// TIA Portal V20 export
FUNCTION_BLOCK "FB_MiscPLC_IHM_ISO"   // FB50, SCL
{ S7_Optimized_Access := 'TRUE' }
// stored: MemoryReserve 100, SetENOAutomatically false
   VAR
      sTransferSelData { S7_SetPoint := 'True'} : Array[0..11] of Byte;
      sTransferActData : Array[0..11] of Byte;
      sUpdate_PLC_ISO_Values : Bool;
      sRT_bStopAfterEmptying : R_TRIG;
      sRT_CNCModeReq { S7_SetPoint := 'True'} : R_TRIG;
   END_VAR
   VAR_TEMP
      tLoop : Int;
      tTransferSelDataError : Int;
      tTransferSelDataErrCode : Array[0..11] of Int;
   END_VAR
BEGIN
   REGION Description header 
       //==================================================================================
       // POSALUX Swiss SA / (C) Copyright 2025
       //----------------------------------------------------------------------------------
       // Title: 
       // Comment/Function: 
       // Author: Fabien WALDT
       // Engineering: TIA Portal v17
       //----------------------------------------------------------------------------------
       // Change log table:
       // Version  | Date     | Expert in charge | Changes applied
       // ---------|----------|------------------|-----------------------------------------
       // 00.00.01 | 20250423 | WFA              | First released version
       // =================================================================================
   END_REGION

   REGION Byte 960
       // Bit 0
       "DB_PLC_ISO_IHM".WarmUpOn := "LBP_AlarmMsgs".UserA[0].A70UUxx[35];

       // Bit 1
       "DB_PLC_ISO_IHM".KeyLaserOn := "DB_DataFromSafety".iKeyLaserOn;

       // Bit 2
       "DB_PLC_ISO_IHM".KeySaveParameters := "DB_McpKeyboardSignals".sK3_KeySaveParam.sKeySWToggleStatus;
       "DB_McpKeyboardSignals".sK3_KeySaveParam.sLedSWStatus := "DB_McpKeyboardSignals".sK3_KeySaveParam.sKeySWToggleStatus;

       // Bit 3
       // STOP_PROG_RUN est nommé bStopAfterEmptying dans PLC
       #sRT_bStopAfterEmptying(CLK := "DB_WorkingModes".sEmptying AND "DB_PartManagement".sPosition.sMachineEmpty);
       IF #sRT_bStopAfterEmptying.Q THEN
           "DB_PLC_ISO_IHM".bStopAfterEmptying := TRUE;
           "LBP_AlarmMsgs".UserA[0].A70UUxx[59] := TRUE;
           "DB_WorkingModes".sEmptying := FALSE;
           "DB_LoaderShuttle1".sMain.iJobReq := FALSE;
           "DB_LoaderShuttle2".sMain.iJobReq := FALSE;
       ELSIF "LBP_Chan1".E_ChanReset THEN
           "DB_PLC_ISO_IHM".bStopAfterEmptying := FALSE;
       END_IF;

       // Bit 4
       "DB_PLC_ISO_IHM".Chan1_running := "DB_CycleStartStop".sChan1Start;

       // Bit 5
       "DB_PLC_ISO_IHM".Chan2_running := FALSE;

       // Bit 6
       "DB_PLC_ISO_IHM".Chan3_running := FALSE;

       // Bit 7
       "DB_PLC_ISO_IHM".Chan4_running := FALSE;
   END_REGION

   REGION Byte 961
       // Bit 0
       "DB_PLC_ISO_IHM".StopAtNextReq := "DB_CycleStartStop".sResquestStopNextCycle;

       // Bit 1
       "DB_PLC_ISO_IHM".AllChanStop := NOT "DB_CycleStartStop".sChan1Start;

       // Bit 2
       "DB_PLC_ISO_IHM".LoaderAutomaticMode := "DB_WorkingModes".sAuto;

       // Bit 3
       "DB_PLC_ISO_IHM".LoaderManualMode := "DB_WorkingModes".sSemiAuto;

       // Bit 4 (NOT USED ON FL0125)
       "DB_PLC_ISO_IHM".NoCameraPresent := "DB_PLC_ISO_IHM".NoCameraPresent;

       // Bit 5 (NOT USED ON FL0125)
       "DB_PLC_ISO_IHM".PremeasureZexists := "DB_PLC_ISO_IHM".PremeasureZexists;

       // Bit 6 (NOT USED ON FL0125)
       "DB_PLC_ISO_IHM".PremeasureCexists := "DB_PLC_ISO_IHM".PremeasureCexists;

       // Bit 7
       "DB_PLC_ISO_IHM".PLCFunctNotFinished :=
       "DB_LoaderFixtureMain".sBlowingNotFinished
       OR "DB_LoaderFixtureMain".sLoadingNotFinished
       OR "DB_LoaderFixtureMain".sUnloadingNotFinished
       OR "DB_LoaderFixtureMain".sReleaseNotFinished
       OR "DB_LoaderFixtureMain".sV_InitNotFinished
       OR "DB_LoaderFixtureMain".sW_InitNotFinished;
   END_REGION

   REGION Byte 962
       // Bit 0
       // CAN_CHANGE_PART_LOADER_1 est nommé StartChangePart_station1 dans PLC
       #sRT_CNCModeReq(CLK := "DB_LoaderAxis".iCNCModeReq);

       IF #sRT_CNCModeReq.Q AND NOT "DB_PartManagement".sPosition.sMachineEmpty THEN
           "DB_PLC_ISO_IHM".StartChangePart_station1 := TRUE;
       ELSIF "LBP_Chan1".MDyn[76] THEN
           "DB_PLC_ISO_IHM".StartChangePart_station1 := FALSE;
       END_IF;

       // Bit 1
       "DB_PLC_ISO_IHM".StartCheckPart_fixture1 := "DB_PLC_ISO_IHM".StartCheckPart_fixture1;

       // Bit 2
       "DB_PLC_ISO_IHM".Loader1PartLoad := "DB_PartManagement".sPosition.sGripper.Undrilled.Presence.Part AND "DB_PartManagement".sPosition.sGripper.Undrilled.Presence.BW;

       // Bit 3
       "DB_PLC_ISO_IHM".Loader1PartUnload := "DB_PartManagement".sPosition.sGripper.Drilled.Presence.Part;

       // Bit 4
       "DB_PLC_ISO_IHM".Loader1ShiftLoad := "DB_PLC_ISO_IHM".Loader1ShiftLoad;

       // Bit 5
       "DB_PLC_ISO_IHM".Loader1ShiftUnload := "DB_PLC_ISO_IHM".Loader1ShiftUnload;

       // Bit 6
       "DB_PLC_ISO_IHM".Loader1LoadOpened := "DB_PLC_ISO_IHM".Loader1LoadOpened;

       // Bit 7
       "DB_PLC_ISO_IHM".Loader1UnloadOpened := "DB_PLC_ISO_IHM".Loader1UnloadOpened;
   END_REGION

   REGION Byte 963
       // Bit 0
       "DB_PLC_ISO_IHM".PartOnFixture1 := "DB_GestionFixture".sFixturePartControl.oGoodPart
               OR "DB_PartManagement".sPosition.sFixture.Undrilled.Presence.Part
               OR "DB_PartManagement".sPosition.sFixture.Drilled.Presence.Part;

       // Bit 1
       "DB_PLC_ISO_IHM".MasterOnFixture1 := "DB_PLC_ISO_IHM".MasterOnFixture1;

       // Bit 2
       "DB_PLC_ISO_IHM".StartChangePart_station2 := "DB_PLC_ISO_IHM".StartChangePart_station2;

       // Bit 3
       "DB_PLC_ISO_IHM".StartCheckPart_fixture2 := "DB_PLC_ISO_IHM".StartCheckPart_fixture2;

       // Bit 4
       "DB_PLC_ISO_IHM".Loader2PartLoad := "DB_PLC_ISO_IHM".Loader2PartLoad;

       // Bit 5
       "DB_PLC_ISO_IHM".Loader2PartUnload := "DB_PLC_ISO_IHM".Loader2PartUnload;

       // Bit 6
       "DB_PLC_ISO_IHM".Loader2ShiftLoad := "DB_PLC_ISO_IHM".Loader2ShiftLoad;

       // Bit 7
       "DB_PLC_ISO_IHM".Loader2ShiftUnload := "DB_PLC_ISO_IHM".Loader2ShiftUnload;
   END_REGION

   REGION Byte 964
       // Bit 0
       "DB_PLC_ISO_IHM".Loader2LoadOpened := "DB_PLC_ISO_IHM".Loader2LoadOpened;

       // Bit 1
       "DB_PLC_ISO_IHM".Loader2UnloadOpened := "DB_PLC_ISO_IHM".Loader2UnloadOpened;

       // Bit 2 
       "DB_PLC_ISO_IHM".PartOnFixture2 := "DB_PLC_ISO_IHM".PartOnFixture2;

       // Bit 3 (NOT USED ON FL0125)
       "DB_PLC_ISO_IHM".MasterOnFixture2 := "DB_PLC_ISO_IHM".MasterOnFixture2;

       // Bit 4 (NOT USED ON FL0125)
       "DB_PLC_ISO_IHM".StartChangePart_station3 := "DB_PLC_ISO_IHM".StartChangePart_station3;

       // Bit 5 (NOT USED ON FL0125)
       "DB_PLC_ISO_IHM".StartCheckPart_fixture3 := "DB_PLC_ISO_IHM".StartCheckPart_fixture3;

       // Bit 6 (NOT USED ON FL0125)
       "DB_PLC_ISO_IHM".Loader3PartLoad := "DB_PLC_ISO_IHM".Loader3PartLoad;

       // Bit 7 (NOT USED ON FL0125)
       "DB_PLC_ISO_IHM".Loader3PartUnload := "DB_PLC_ISO_IHM".Loader3PartUnload;
   END_REGION

   REGION Byte 965
       // Bit 0 (NOT USED ON FL0125)
       "DB_PLC_ISO_IHM".Loader3ShiftLoad := "DB_PLC_ISO_IHM".Loader3ShiftLoad;

       // Bit 1 (NOT USED ON FL0125)
       "DB_PLC_ISO_IHM".Loader3ShiftUnload := "DB_PLC_ISO_IHM".Loader3ShiftUnload;

       // Bit 2 (NOT USED ON FL0125)
       "DB_PLC_ISO_IHM".Loader3LoadOpened := "DB_PLC_ISO_IHM".Loader3LoadOpened;

       // Bit 3
       "DB_PLC_ISO_IHM".Loader3UnloadOpened := "DB_PLC_ISO_IHM".Loader3UnloadOpened;

       // Bit 4
       "DB_PLC_ISO_IHM".PartOnFixture3 := "DB_PLC_ISO_IHM".PartOnFixture3;

       // Bit 5 (NOT USED ON FL0125)
       "DB_PLC_ISO_IHM".MasterOnFixture3 := "DB_PLC_ISO_IHM".MasterOnFixture3;

       // Bit 6 (NOT USED ON FL0125)
       "DB_PLC_ISO_IHM".Part_KO_go_outside_mach := "DB_PLC_ISO_IHM".Part_KO_go_outside_mach;

       // Bit 7 (NOT USED ON FL0125)
       "DB_PLC_ISO_IHM".MasterOnMachine := "DB_PLC_ISO_IHM".MasterOnMachine;
   END_REGION

   REGION Word 968
       "DB_PLC_ISO_IHM".WarmUpTime := "DB_PLC_ISO_IHM".WarmUpTime;
   END_REGION

   REGION Byte 970
       // Bit 0
       "DB_PLC_ISO_IHM".Stop_For_BackWall_Wear_1 := "DB_PLC_ISO_IHM".Stop_For_BackWall_Wear_1;

       // Bit 1
       "DB_PLC_ISO_IHM".Stop_For_BackWall_Wear_2 := "DB_PLC_ISO_IHM".Stop_For_BackWall_Wear_2;

       // Bit 2
       "DB_PLC_ISO_IHM".Cleaning_Station_1 := "DB_PLC_ISO_IHM".Cleaning_Station_1;

       // Bit 3
       "DB_PLC_ISO_IHM".Cleaning_Station_2 := "DB_PLC_ISO_IHM".Cleaning_Station_2;

       // Bit 4
       "DB_PLC_ISO_IHM".Cleaning_Backwall_1 := "DB_PLC_ISO_IHM".Cleaning_Backwall_1;

       // Bit 5
       "DB_PLC_ISO_IHM".Cleaning_Backwall_2 := "DB_PLC_ISO_IHM".Cleaning_Backwall_2;

       // Bit 6
       "DB_PLC_ISO_IHM".Shutter_laser_closed := "DB_DigitalInputs".sShutterClosed.sSWStatus OR
            NOT "DB_DataFromSafety".iKeyLaserOn;

       // Bit 7
       "DB_PLC_ISO_IHM".Pressure_Stop_Machine := "DB_PLC_ISO_IHM".Pressure_Stop_Machine;
   END_REGION

   REGION Byte 971  
       // Bit 0
       IF "LBP_Chan1".MDyn[68] OR "DB_Scanner".sScannerComm.oGoodPart THEN
           "DB_PLC_ISO_IHM".BadPartOnFixture := FALSE;
       ELSIF "DB_BadPartOnFixture".BadPartOnFixture
           OR "DB_GestionFixture".sFixturePartControl.oBadpart
           OR "DB_Scanner".sScannerComm.oBadPart THEN
               "DB_PLC_ISO_IHM".BadPartOnFixture := TRUE;
       END_IF;

       // Bit 1 (NOT USED ON FL0125)
       "DB_PLC_ISO_IHM".Reserve12 := "DB_PLC_ISO_IHM".Reserve12;

       // Bit 2 (NOT USED ON FL0125)
       "DB_PLC_ISO_IHM".Reserve13 := "DB_PLC_ISO_IHM".Reserve13;

       // Bit 3 (NOT USED ON FL0125)
       "DB_PLC_ISO_IHM".Reserve14 := "DB_PLC_ISO_IHM".Reserve14;

       // Bit 4 (NOT USED ON FL0125)
       "DB_PLC_ISO_IHM".Reserve15 := "DB_PLC_ISO_IHM".Reserve15;

       // Bit 5
       "DB_PLC_ISO_IHM".SemiAuto_RunEmpty := "DB_PLC_ISO_IHM".SemiAuto_RunEmpty;

       // Bit 6
       "DB_PLC_ISO_IHM"."SemiAuto_Unload_C-Fixture" := "DB_PLC_ISO_IHM"."SemiAuto_Unload_C-Fixture";

       // Bit 7 (NOT USED ON FL0125)
       "DB_PLC_ISO_IHM".Reserve18 := "DB_PLC_ISO_IHM".Reserve18;
   END_REGION

   REGION Transfert data PLC -> ISO

       FOR #tLoop := 0 TO 11 DO
           #sTransferActData[#tLoop] := PEEK(area := 16#84, dbNumber := 1302, byteOffset := #tLoop);
           IF #sTransferActData[#tLoop] <> #sTransferSelData[#tLoop] THEN
               #sUpdate_PLC_ISO_Values := TRUE;
               #sTransferSelData[#tLoop] := #sTransferActData[#tLoop];
           END_IF;
       END_FOR;

       // Transfert DB_PLC_ISO_IHM DWORD 0  

       // DEFINE PART_ON_FIXTURE_1         AS (($A_DBB[963] B_AND 1)==1)
       // DEFINE MASTER_ON_FIXTURE_1       AS (($A_DBB[963] B_AND 2)==2)
       // DEFINE CAN_CHANGE_PART_LOADER_2  AS (($A_DBB[963] B_AND 4)==4)
       // DEFINE CHECK_PART_FIXTURE_2      AS (($A_DBB[963] B_AND 8)==8)
       // DEFINE LOADER_2_PART_LOAD        AS (($A_DBB[963] B_AND 16)==16)
       // DEFINE LOADER_2_PART_UNLOAD      AS (($A_DBB[963] B_AND 32)==32)
       // DEFINE LOADER_2_SHIFT_LOAD       AS (($A_DBB[963] B_AND 64)==64)
       // DEFINE LOADER_2_SHIFT_UNLOAD     AS (($A_DBB[963] B_AND 128)==128)

       "LBP_TransferSelData"(Enable := #sUpdate_PLC_ISO_Values,
                             Funct := BYTE#16#04,
                             IVAR1 := 963,
                             IVAR2 := -1,
                             Error => #tTransferSelDataError.%X0,
                             ErrCode => #tTransferSelDataErrCode[0],
                             S7Var := #sTransferSelData[3]);

       // DEFINE CAN_CHANGE_PART_LOADER_1  AS (($A_DBB[962] B_AND 1)==1)
       // DEFINE CHECK_PART_FIXTURE_1      AS (($A_DBB[962] B_AND 2)==2)
       // DEFINE LOADER_1_PART_LOAD        AS (($A_DBB[962] B_AND 4)==4)
       // DEFINE LOADER_1_PART_UNLOAD      AS (($A_DBB[962] B_AND 8)==8)
       // DEFINE LOADER_1_SHIFT_LOAD       AS (($A_DBB[962] B_AND 16)==16)
       // DEFINE LOADER_1_SHIFT_UNLOAD     AS (($A_DBB[962] B_AND 32)==32)
       // DEFINE LOADER_1_LOAD_OPENED      AS (($A_DBB[962] B_AND 64)==64)
       // DEFINE LOADER_1_UNLOAD_OPENED    AS (($A_DBB[962] B_AND 128)==128)

       "LBP_TransferSelData"(Enable := #sUpdate_PLC_ISO_Values,
                             Funct := BYTE#16#04,
                             IVAR1 := 962,
                             IVAR2 := -1,
                             Error => #tTransferSelDataError.%X1,
                             ErrCode => #tTransferSelDataErrCode[1],
                             S7Var := #sTransferSelData[2]);

       // DEFINE STOP_AT_NEXT_REQ          AS (($A_DBB[961] B_AND 1)==1)
       // DEFINE ALL_CHAN_STOP             AS (($A_DBB[961] B_AND 2)==2)
       // DEFINE LOADER_MODE_AUTOMATIC     AS (($A_DBB[961] B_AND 4)==4)
       // DEFINE LOADER_MODE_MANUAL        AS (($A_DBB[961] B_AND 8)==8)
       // DEFINE MODE_WITH_LOADER          AS (($A_DBB[961] B_AND 12)>0)
       // DEFINE MODE_WITHOUT_LOADER       AS (($A_DBB[961] B_AND 12)==0)
       // DEFINE NO_CAMERA_PRESENT         AS (($A_DBB[961] B_AND 16)==16)
       // DEFINE PREMEASURE_Z_EXISTS       AS (($A_DBB[961] B_AND 32)==32)
       // DEFINE PREMEASURE_C_EXISTS       AS (($A_DBB[961] B_AND 64)==64)

       "LBP_TransferSelData"(Enable := #sUpdate_PLC_ISO_Values,
                             Funct := BYTE#16#04,
                             IVAR1 := 961,
                             IVAR2 := -1,
                             Error => #tTransferSelDataError.%X2,
                             ErrCode => #tTransferSelDataErrCode[2],
                             S7Var := #sTransferSelData[1]);

       // DEFINE WARM_UP_ON                AS (($A_DBB[960] B_AND 1)==1)
       // DEFINE KEY_LASER_ON              AS (($A_DBB[960] B_AND 2)==2)
       // DEFINE KEY_SAVE_PARAM            AS (($A_DBB[960] B_AND 4)==4)
       // DEFINE STOP_PROG_RUN             AS (($A_DBB[960] B_AND 8)==8)
       // DEFINE CHAN_1_RUNNING            AS (($A_DBB[960] B_AND 16)==16)
       // DEFINE CHAN_2_RUNNING            AS (($A_DBB[960] B_AND 32)==32)
       // DEFINE CHAN_3_RUNNING            AS (($A_DBB[960] B_AND 64)==64)
       // DEFINE CHAN_4_RUNNING            AS (($A_DBB[960] B_AND 128)==128)

       "LBP_TransferSelData"(Enable := #sUpdate_PLC_ISO_Values,
                             Funct := BYTE#16#04,
                             IVAR1 := 960,
                             IVAR2 := -1,
                             Error => #tTransferSelDataError.%X3,
                             ErrCode => #tTransferSelDataErrCode[3],
                             S7Var := #sTransferSelData[0]);

       // Transfert DB_PLC_ISO_IHM DWORD 4  


       "LBP_TransferSelData"(Enable := #sUpdate_PLC_ISO_Values,
                             Funct := BYTE#16#04,
                             IVAR1 := 967,
                             IVAR2 := -1,
                             Error => #tTransferSelDataError.%X4,
                             ErrCode => #tTransferSelDataErrCode[4],
                             S7Var := #sTransferSelData[7]);

       "LBP_TransferSelData"(Enable := #sUpdate_PLC_ISO_Values,
                             Funct := BYTE#16#04,
                             IVAR1 := 966,
                             IVAR2 := -1,
                             Error => #tTransferSelDataError.%X5,
                             ErrCode => #tTransferSelDataErrCode[5],
                             S7Var := #sTransferSelData[6]);

       // DEFINE LOADER_3_SHIFT_LOAD       AS (($A_DBB[965] B_AND 1)==1)
       // DEFINE LOADER_3_SHIFT_UNLOAD     AS (($A_DBB[965] B_AND 2)==2)
       // DEFINE LOADER_3_LOAD_OPENED      AS (($A_DBB[965] B_AND 4)==4)
       // DEFINE LOADER_3_UNLOAD_OPENED    AS (($A_DBB[965] B_AND 8)==8)
       // DEFINE PART_ON_FIXTURE_3         AS (($A_DBB[965] B_AND 16)==16)
       // DEFINE MASTER_ON_FIXTURE_3       AS (($A_DBB[965] B_AND 32)==32)
       // DEFINE PART_KO_GO_OUTSIDE        AS (($A_DBB[965] B_AND 64)==64)
       // DEFINE MASTER_ON_MACHINE         AS (($A_DBB[965] B_AND 128)==128)

       "LBP_TransferSelData"(Enable := #sUpdate_PLC_ISO_Values,
                             Funct := BYTE#16#04,
                             IVAR1 := 965,
                             IVAR2 := -1,
                             Error => #tTransferSelDataError.%X6,
                             ErrCode => #tTransferSelDataErrCode[6],
                             S7Var := #sTransferSelData[5]);

       // DEFINE LOADER_2_LOAD_OPENED      AS (($A_DBB[964] B_AND 1)==1)
       // DEFINE LOADER_2_UNLOAD_OPENED    AS (($A_DBB[964] B_AND 2)==2)
       // DEFINE PART_ON_FIXTURE_2         AS (($A_DBB[964] B_AND 4)==4)
       // DEFINE MASTER_ON_FIXTURE_2       AS (($A_DBB[964] B_AND 8)==8)
       // DEFINE CAN_CHANGE_PART_LOADER_3  AS (($A_DBB[964] B_AND 16)==16)
       // DEFINE CHECK_PART_FIXTURE_3      AS (($A_DBB[964] B_AND 32)==32)
       // DEFINE LOADER_3_PART_LOAD        AS (($A_DBB[964] B_AND 64)==64)
       // DEFINE LOADER_3_PART_UNLOAD      AS (($A_DBB[964] B_AND 128)==128)

       "LBP_TransferSelData"(Enable := #sUpdate_PLC_ISO_Values,
                             Funct := BYTE#16#04,
                             IVAR1 := 964,
                             IVAR2 := -1,
                             Error => #tTransferSelDataError.%X7,
                             ErrCode => #tTransferSelDataErrCode[7],
                             S7Var := #sTransferSelData[4]);

       // Transfert DB_PLC_ISO_IHM DWORD 8  

       // DEFINE SET_BAD_PART_ON_FIXTURE   AS (($A_DBB[971] B_AND 1)==1)
       // ;DEFINE     AS (($A_DBB[971] B_AND 2)==2)
       // ;DEFINE     AS (($A_DBB[971] B_AND 4)==4)
       // ;DEFINE     AS (($A_DBB[971] B_AND 8)==8)
       // ;DEFINE     AS (($A_DBB[971] B_AND 16)==16)
       // DEFINE SEMIAUTO_RUNEMPTY         AS (($A_DBB[971] B_AND 32)==32)
       // DEFINE SEMIAUTO_UNLOAD_C_FIXTURE AS (($A_DBB[971] B_AND 64)==64)
       // ;DEFINE     AS (($A_DBB[971] B_AND 128)==128

       "LBP_TransferSelData"(Enable := #sUpdate_PLC_ISO_Values,
                             Funct := BYTE#16#04,
                             IVAR1 := 971,
                             IVAR2 := -1,
                             Error => #tTransferSelDataError.%X8,
                             ErrCode => #tTransferSelDataErrCode[8],
                             S7Var := #sTransferSelData[11]);

       // DEFINE STOP_FOR_BACKWALL1_WEARED AS (($A_DBB[970] B_AND 1)==1)
       // DEFINE STOP_FOR_BACKWALL2_WEARED AS (($A_DBB[970] B_AND 2)==2)
       // DEFINE CLEANING_STATION1         AS (($A_DBB[970] B_AND 4)==4)
       // DEFINE CLEANING_STATION2         AS (($A_DBB[970] B_AND 8)==8)
       // DEFINE CLEANING_BACKWALL1        AS (($A_DBB[970] B_AND 16)==16)
       // DEFINE CLEANING_BACKWALL2        AS (($A_DBB[970] B_AND 32)==32)
       // DEFINE LASER_SHUTTER_CLOSED      AS (($A_DBB[970] B_AND 64)==64)
       // DEFINE NOT_COND_FOR_DRILL        AS (($A_DBB[970] B_AND 128)==128)

       "LBP_TransferSelData"(Enable := #sUpdate_PLC_ISO_Values,
                             Funct := BYTE#16#04,
                             IVAR1 := 970,
                             IVAR2 := -1,
                             Error => #tTransferSelDataError.%X9,
                             ErrCode => #tTransferSelDataErrCode[9],
                             S7Var := #sTransferSelData[10]);


       "LBP_TransferSelData"(Enable := #sUpdate_PLC_ISO_Values,
                             Funct := BYTE#16#04,
                             IVAR1 := 969,
                             IVAR2 := -1,
                             Error => #tTransferSelDataError.%X10,
                             ErrCode => #tTransferSelDataErrCode[10],
                             S7Var := #sTransferSelData[9]);

       // DEFINE WARM_UP_TIME              AS ($A_DBW[968])

       "LBP_TransferSelData"(Enable := #sUpdate_PLC_ISO_Values,
                             Funct := BYTE#16#04,
                             IVAR1 := 968,
                             IVAR2 := -1,
                             Error => #tTransferSelDataError.%X11,
                             ErrCode => #tTransferSelDataErrCode[11],
                             S7Var := #sTransferSelData[8]);

       IF #tTransferSelDataError = 0 THEN
           #sUpdate_PLC_ISO_Values := FALSE;
       END_IF;
   END_REGION
END_FUNCTION_BLOCK
